{attribute 'no_explicit_call' := 'do not call this POU directly'} 
FUNCTION_BLOCK FB_ListObject IMPLEMENTS I_ListObject
VAR
	pList: 			POINTER TO I_Object;
	{IF (defined (release))}
    	{attribute 'hide'}
	{END_IF}
	aList:			POINTER TO POINTER TO ARRAY [0..24] OF I_Object:=ADR(pList);
END_VAR
VAR_OUTPUT
	{IF (defined (release))}
    	{attribute 'hide'}
	{END_IF}
	nLength:		INT;	
END_VAR

// https://peterzerlauth.com/

METHOD FB_exit : BOOL
VAR_INPUT
	bInCopyCode : BOOL; // if TRUE, the exit method is called for exiting an instance that is copied afterwards (online change).
END_VAR
M_Clear();
END_METHOD

METHOD PUBLIC M_Add : BOOL
VAR_INPUT
	Object: 	I_Object;
END_VAR
VAR
	pOldList: 	POINTER TO I_Object;
END_VAR
IF Object <> 0 THEN
	// First Item
	IF pList = 0 THEN
		nLength:= nLength + 1;
		pList:= __NEW(POINTER TO I_Object,DINT_TO_UDINT(nLength));
	ELSE
		// Item already in List
		IF M_Find(Object) = -1 THEN
			// backup 
			pOldList:= pList;
			// new Length
			nLength:= nLength + 1;
			// new pointer
			pList:= __NEW(POINTER TO I_Object,DINT_TO_UDINT(nLength));
			// restore
			Memcpy(pList,pOldList, SIZEOF(POINTER TO I_Object)*DINT_TO_UDINT(nLength -1));
			// delete old
			__DELETE(pOldList);
		ELSE
			M_Add:= FALSE;	
			RETURN;
		END_IF
	END_IF
	IF pList = 0 THEN
		RETURN;
	END_IF
	// add new Object
	pList[nLength-1]:= Object;
	M_Add:= TRUE;
ELSE
	M_Add:= FALSE;	
END_IF
END_METHOD

METHOD PUBLIC M_Clear : bool
IF pList <> 0 THEN
	nLength:= 0;
	__DELETE(pList);
END_IF
M_Clear:= TRUE;
END_METHOD

METHOD PUBLIC M_Find : DINT
VAR_INPUT
	Object: 	I_Object;
END_VAR
VAR
	nIndex: 	UINT;
END_VAR
// Object already in List
M_Find := -1;
WHILE nIndex < nLength DO
    IF (pList[nIndex] = Object) THEN
        M_Find := nIndex;
        RETURN;
    END_IF
	nIndex := nIndex + 1;
END_WHILE
END_METHOD

METHOD PUBLIC M_Index : I_Object
VAR_INPUT
	Index: 	DINT;
END_VAR
IF Index <= nLength THEN
	M_Index:= pList[Index];
END_IF
END_METHOD

METHOD PUBLIC M_Remove : BOOL
VAR_INPUT
	Object: 	I_Object;
END_VAR
VAR
	pOldList:			POINTER TO I_Object;
	nPosition: 			DINT;
END_VAR
IF Object <> 0 THEN
	// First Item
	IF nLength >= 0 THEN
		// Item already in List
		nPosition:= M_Find(Object);
		IF nPosition <> -1 THEN
			// backup 
			pOldList:= pList;
			// new Length
			nLength:= nLength -1;
			// new pointer
			pList:= __NEW(POINTER TO I_Object,DINT_TO_UDINT(nLength));
			// restore lower part
			Memcpy(pList,pOldList, SIZEOF(POINTER TO I_Object) * DINT_TO_UDINT(nPosition));
			//pList[nPosition]:= iObject;
			Memcpy(pList + (SIZEOF(POINTER TO I_Object)*nPosition),pOldList + (SIZEOF(POINTER TO I_Object)*(nPosition + 1)), SIZEOF(POINTER TO I_Object) * DINT_TO_UDINT(nLength - nPosition));
			// delete old
			__DELETE(pOldList);
		ELSE
			M_Remove:= FALSE;	
			RETURN;
		END_IF
	ELSE
		M_Remove:= FALSE;	
		RETURN;
	END_IF
	M_Remove:= TRUE;
ELSE
	M_Remove:= FALSE;	
END_IF
END_METHOD

{attribute 'OPC.UA.DA.Property' := '1'}
{attribute 'monitoring' := 'call'}
PROPERTY PUBLIC P_Length : DINT
GET
P_Length:= nLength;
END_GET
END_PROPERTY

END_FUNCTION_BLOCK

(* stored: Version 1.1.0.1
   POU FB_ListObject: Id {9081e76d-9be0-4c60-ba53-64a67cdcc01f}, SpecialFunc None
   Method FB_exit: Id {7daa207b-cd6f-4003-b787-3b64334babbc}
   Method M_Add: Id {573e88b0-086d-4607-8280-9e200d874ce5}
   Method M_Clear: Id {5185d8d5-9632-41dd-9f2f-711936332e5b}
   Method M_Find: Id {4c0f1cf5-9a17-45e4-a85a-c781ed972a27}
   Method M_Index: Id {919bdfbb-db0e-4a7f-8ca8-f758ff962a94}
   Method M_Remove: Id {e9807c5c-b966-4419-87bc-84d068abfb2d}
   Property P_Length: Id {d45b982f-4b97-465f-bb53-55cc6ad8a8d4}
   Get Get: Id {9d0b7376-3a4d-4a08-aa02-0d3f8f110cdd} *)
